FUNCTION MultiplicationFunction : REAL
VAR_INPUT
	i_rValueA : REAL;
	i_rValueB : REAL;
END_VAR
VAR
END_VAR

MultiplicationFunction := i_rValueA * i_rValueB;

END_FUNCTION

(* stored: Version 1.1.0.1, ProductVersion 3.1.4022.12
   POU MultiplicationFunction: Id {1465d7da-c6a2-49b6-b9f6-cb9bf527f1ef}, SpecialFunc None *)
